RoboDK station: hans_e10l_assembled_colored_industrial.rdk

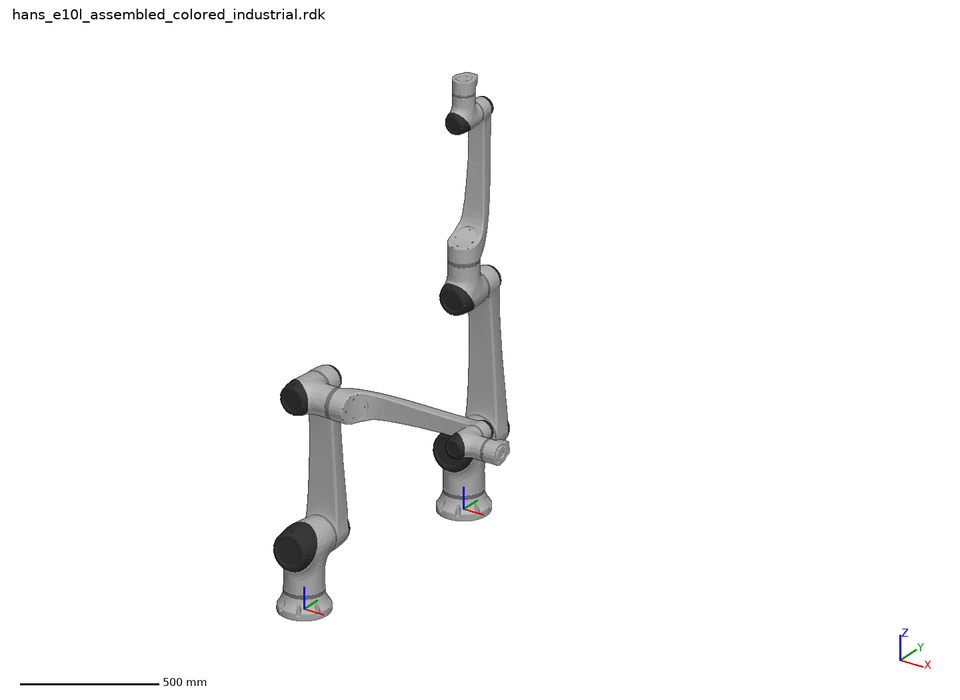
[picture v0: the station drawn from its stored meshes, robots at their saved joint values, targets as dots, program paths as lines]
Station hans_e10l (saved by RoboDK 5.4.0). Poses are relative to the parent item; angles as X-Y-Z fixed-axis rotations.
  - frame Hans E10L Base at (0, 0, 0) mm
    - object link_0 at (0, 0, 0) mm, size 192.7 x 200 x 77.5 mm
    - object link_1 at (0, 0, 0) mm, size 166.1 x 210.2 x 271.5 mm
    - object link_2 at (0, 0, 0) mm, size 152 x 115.1 x 735.7 mm
    - object link_3 at (0, 0, 0) mm, size 223.5 x 179.1 x 129 mm
    - object link_4 at (0, 0, 0) mm, size 596.8 x 195.6 x 120 mm
    - object link_5 at (0, 0, 0) mm, size 157 x 149.6 x 92.4 mm
    - object link_6 at (0, 0, 0) mm, size 57.5 x 102.5 x 85 mm
  - frame Han's E10L Base at (0, 1000, 0) mm
    - robot Han's E10L: 6 axes
        modified DH rows (alpha deg, a mm, theta deg, d mm): 0, 0, 0, 260; -90, 0, -90, 0; 0, 600, -90, 0; -90, 0, 0, 700; 90, 0, 0, 0; -90, 0, 180, 168
        joint limits [-180, -170, -170, -180, -180, -360] to [180, 170, 170, 180, 180, 360]; home [0, 0, 0, 0, 0, 0]; saved at [0, 0, 0, 0, 0, 0]
